{attribute 'hide_all_locals'}
(* 用于在多种常用的时间格式间进行转换的功能块,不考虑时区 *)
FUNCTION_BLOCK FB_TimeConvertorM_1
VAR_INPUT
	InputType : UDINT := 0 ; (* 0:DcTaskTime 1:10位Unix 2:13位Unix 3:FileTime64 4:DateAndTime 5:SystemTime *)
	iDcTaskTime : LINT; (* DcTaskTime从2000-01-01 00:00:00:000开始，精确到1ns *)
	iUnixTimeStamp10 : ULINT; (* 10位unix时间戳，代表从格林威治时间1970-01-01 00:00:00开始的秒数 *)
	iUnixTimeStamp13 : ULINT; (* 13位unix时间戳，代表从格林威治时间1970-01-01 00:00:00开始的秒数+3位毫秒数 *)
	iFileTime64 : T_FILETIME64; (* Utilities库中引入的Windows文件系统时间戳，代表从格林威治时间1601-01-01 00:00:00开始的纳秒数 *)
	iDateAndTime : DATE_AND_TIME; (* TwinCAT系统自带的本地时间日期格式，数值为10位unix时间戳，受到时区影响 *)
	iSystemTime : TIMESTRUCT; (* Utilities库中定义的本地时间日期格式，包含了年月日时分秒毫秒的结构体，受到时区影响 *)
END_VAR
VAR_OUTPUT
	oDcTaskTime : LINT;(* DcTaskTime从2000-01-01 00:00:00:000开始，精确到1ns *)
	oUnixTimeStamp10 : ULINT; (* 10位unix时间戳，代表从格林威治时间1970-01-01 00:00:00开始的秒数 *)
	oUnixTimeStamp13 : ULINT; (* 13位unix时间戳，代表从格林威治时间1970-01-01 00:00:00开始的秒数+3位毫秒数 *)
	oFileTime64 : T_FILETIME64; (* Utilities库中引入的Windows文件系统时间戳，代表从格林威治时间1601-01-01 00:00:00开始的纳秒数 *)
	oDateAndTime : DATE_AND_TIME; (* TwinCAT系统自带的本地时间日期格式，数值为10位unix时间戳，受到时区影响 *)
	oSystemTime : TIMESTRUCT; (* Utilities库中定义的本地时间日期格式，包含了年月日时分秒毫秒的结构体，受到时区影响 *)
	oStringTime : STRING(23); (* 时间字符串，年月日时分秒毫秒 *)
	oStringDate : STRING(10); (* 时间字符串，年月日 *)
	oStringTimeOfDay : STRING(12); (* 时间字符串，时分秒毫秒 *)
END_VAR
VAR
END_VAR

(* 测试数据751214127491000000,1697898927,1697898927491,LDT#2023-10-21-14:35:22.491,DT#2023-10-21-14:35:22,..  *)
(* 由于Utilities库中自带了Filetime64与DT, Systemtime之间的转换，本功能块仅仅是添加了Filetime64与DcTaskTime与UnixTimeStamp之前的转换 *)
(* 转换思路是先尽可能转换成Filetime64，再利用自带函数转换 *)
(* Filetime64与DcTaskTime与UnixTimeStamp都是一种时间戳，区别在于起始时间或精度各不相同 *)
(* DcTaskTime从2000-01-01 00:00:00:000开始，精确到1ns *)
(* 10位Unix时间戳从1970-01-01 00:00:00开始，精确到1s，13位Unix时间戳加了三位表示毫秒的数 *)
(* FileTime64从1601-01-01 00:00:00开始，精确到100ns, *)
(* 946684800:从1970-2000年的秒数  11644473600:从1601-1970的秒数  5:误差补偿 *)
CASE InputType OF
	0:(* DcTaskTime从2000-01-01 00:00:00:000开始，精确到1ns *)
	(* Input *)
	oDcTaskTime := iDcTaskTime;
	(* Convert *)
	oFileTime64 := LINT_TO_ULINT(oDcTaskTime)/100 + 946684800_0000000 + 11644473600_0000000 - 5_0000000;
	oUnixTimeStamp13 := oFileTime64/10000 + 5000 - 11644473600000;
	oUnixTimeStamp10 := oUnixTimeStamp13 / 1000;
	oDateAndTime := FILETIME64_TO_DT(oFileTime64);
	oSystemTime := FILETIME64_TO_SYSTEMTIME(oFileTime64);
	
	1: (* Unix10 -> Unix13 : 由于10位时间戳不包含毫秒，所以转换出来的也不包含 *)
	(* Input *)
	oUnixTimeStamp10 := iUnixTimeStamp10;
	(* Convert *)
	oUnixTimeStamp13 := oUnixTimeStamp10 * 1000;
	oFileTime64 := (oUnixTimeStamp13 + 11644473600000 - 5000) * 10000;
	oDateAndTime := FILETIME64_TO_DT(oFileTime64);
	oSystemTime := FILETIME64_TO_SYSTEMTIME(oFileTime64);
	oDcTaskTime := ULINT_TO_LINT(oFileTime64 - 946684800_0000000 - 11644473600_0000000 + 5_0000000) * 100;
	
	2:
	(* Input *)
	oUnixTimeStamp13 := iUnixTimeStamp13;
	(* Convert *)
	oUnixTimeStamp10 := oUnixTimeStamp13 / 1000;
	oFileTime64 := (oUnixTimeStamp13 + 11644473600000 - 5000) * 10000;
	oDateAndTime := FILETIME64_TO_DT(oFileTime64);
	oSystemTime := FILETIME64_TO_SYSTEMTIME(oFileTime64);
	oDcTaskTime := ULINT_TO_LINT(oFileTime64 - 946684800_0000000 - 11644473600_0000000 + 5_0000000) * 100;
	
	3:
	(* Input *)
	oFileTime64 := iFileTime64;
	(* Convert *)
	oUnixTimeStamp13 := oFileTime64/10000 + 5000 - 11644473600000;
	oUnixTimeStamp10 := oUnixTimeStamp13 / 1000;
	oDateAndTime := FILETIME64_TO_DT(oFileTime64);
	oSystemTime := FILETIME64_TO_SYSTEMTIME(oFileTime64);
	oDcTaskTime := ULINT_TO_LINT(oFileTime64 - 946684800_0000000 - 11644473600_0000000 + 5_0000000) * 100;
	
	4:
	(* Input *)
	oDateAndTime := iDateAndTime;
	(* Convert *)
	oFileTime64 := DT_TO_FILETIME64(oDateAndTime);
	oUnixTimeStamp13 := oFileTime64/10000 + 5000 - 11644473600000;
	oUnixTimeStamp10 := oUnixTimeStamp13 / 1000;
	oSystemTime := FILETIME64_TO_SYSTEMTIME(oFileTime64);
	oDcTaskTime := ULINT_TO_LINT(oFileTime64 - 946684800_0000000 - 11644473600_0000000 + 5_0000000) * 100;
	
	5:
	(* Input *)
	oSystemTime :=iSystemTime;
	(* Convert *)
	oFileTime64 := SYSTEMTIME_TO_FILETIME64(oSystemTime);
	oUnixTimeStamp13 := oFileTime64/10000 + 5000 - 11644473600000;
	oUnixTimeStamp10 := oUnixTimeStamp13 / 1000;
	oDateAndTime := FILETIME64_TO_DT(oFileTime64);
	oDcTaskTime := ULINT_TO_LINT(oFileTime64 - 946684800_0000000 - 11644473600_0000000 + 5_0000000) * 100;
	
END_CASE
(* 2023-10-21 15:18:31:771 *)
oStringTime := F_SYSTEMTIME_TO_String6(oSystemTime, '');
oStringDate := MID(STR:= oStringTime, LEN:= 10, POS:= 1);
oStringTimeOfDay := MID(STR:= oStringTime, LEN:= 12, POS:= 12);

END_FUNCTION_BLOCK

(* stored: Version 1.1.0.1, ProductVersion 3.1.4024.12
   POU FB_TimeConvertorM_1: Id {eb28e114-3ef9-4ec4-b7ac-1369c7907dac}, SpecialFunc None *)
